INTERFACE I_Pid

METHOD Reset
END_METHOD

METHOD Update : LREAL
VAR_INPUT
    fSetpoint    : LREAL;
    fMeasurement : LREAL;
    fDeltaT      : LREAL;
END_VAR
END_METHOD

END_INTERFACE

(* stored: Version 1.1.0.1
   Itf I_Pid: Id {b5e48d33-99a7-455a-9a71-25c357c0c781}
   Method Reset: Id {3a74c138-43f7-4dde-9295-168397c146fe}
   Method Update: Id {12494460-92f3-43f3-b78c-78528912bf97} *)
